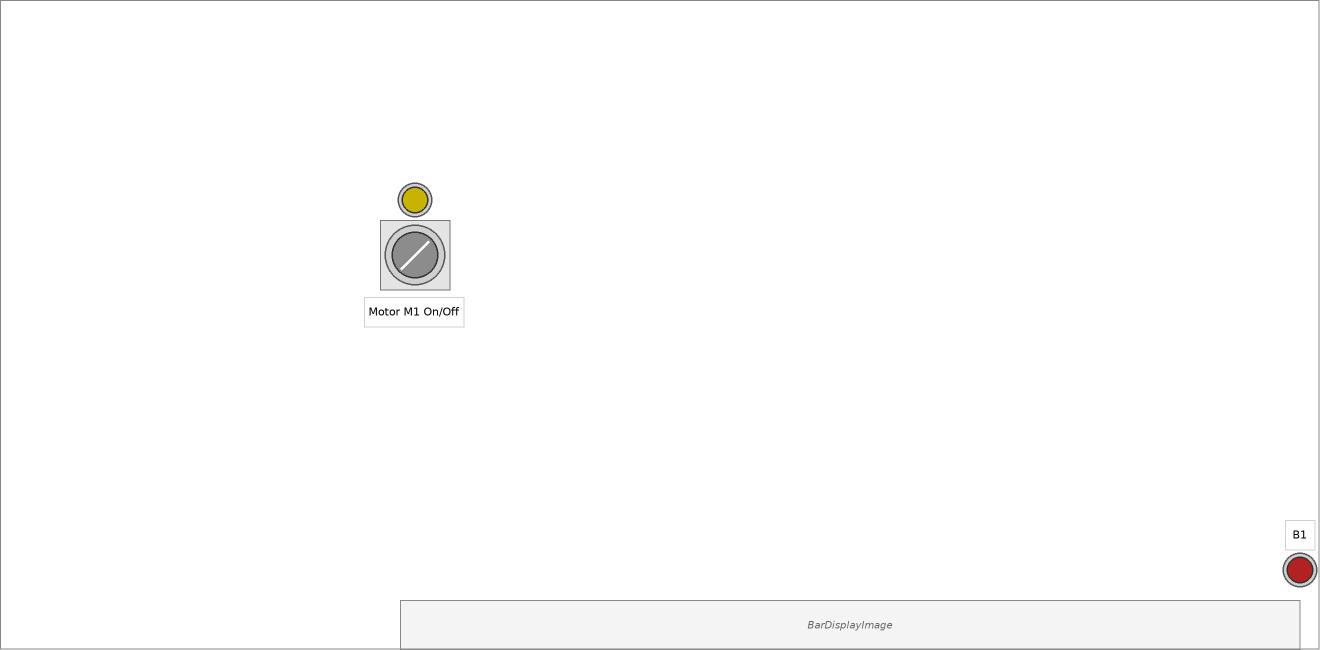
VISUALIZATION Visualization  // 1320x650
VAR_IN_OUT
END_VAR
//Palkki ei liiku, lisää napit paketin laittamiselle ja poistamiselle
    BarDisplayImage (400,600 900x50), value: GVL._TimeOnConveyor, style: BarDisplayImage-Blue, scale format: %.1f, scale 0..100
    RotarySwitch (380,220 70x70), variable: GVL._Switch, behaviour: TOGGLE, style: Switch-RotarySwitch-Gray
    Lamp1 (1280,550 40x40), variable: GVL._SensorCovered, style: Lamp-Lamp1-Red
    Textfield (1285,520 30x30), "B1"
    Textfield (364,297 100x30), "Motor M1 On/Off"
    Lamp1 (395,180 40x40), variable: GVL._Switch, style: Lamp-Lamp1-Yellow
END_VISUALIZATION

(* stored: Version 1.1.0.1
   Visu Visualization: Id {d1484e27-88de-4ca3-b2cf-aa90e81c1ce2} *)
